{attribute 'qualified_only'}
TYPE LinearAxis_e :
(
    ST110_01Y,
    ST110_02Z,
    ST110_03Z,
    ST110_04Z,
    ST115_01Y,
    ST115_02Z,
    ST115_03Z,
    ST115_04Z,
    ST120_01Y,
    ST120_02Z,
    ST125_01Y,
    ST125_02Z,
	ST130_01Z,
	ST130_10Z,
	ST135_01Z,
	ST135_10Z,
	ST145_01Y,
	ST145_02Z,
	ST160_01Z,
	ST165_01Z,
	ST170_01Z,
	ST180_01Y,
	ST180_02Z,
	ST180_10Z,
	ST185_01Y,
	ST185_02Z,
	ST185_10Z,
    _max
);
END_TYPE

(* stored: Version 1.1.0.1, ProductVersion 3.1.4024.6
   EnumerationTextList LinearAxis_e: Id {de49f3bc-7d80-4b86-8b23-defa93556e22} *)
